// TIA Portal V21 export
TYPE "Rcp_Capper"
   STRUCT
      Abilitazione : Bool;   // Tappatore abilitato
      AltezzaCarosello : Real;
      TipoDiTappo : Int;
      VelocitàBassaOrientatoreTappi : Real;
      VelocitàAltaOrientatoreTappi : Real;
      VelocitàVibratoreTappiElevatore : Real;
      VelocitàElevatoreTappi : Real;
      VelocitàNastroTappi : Real;
   END_STRUCT;
END_TYPE
